// TIA Portal project "Project_Benzinarie" (V15.1)

(* hardware
DEVICE "S71500/ET200MP station_1"  S7-1500 station
   slot 0: "Rail_0"  Rack  6ES7 590-1***0-0AA0
   slot 1: "PLC_1"  CPU 1513-1 PN  6ES7 513-1AL02-0AB0  V2.6
      slot 3: "CPU display_1"  6ES7591-1AA00-0AA0
*)

// ===== PLC "PLC_1"  CPU 1513-1 PN =====

VAR_GLOBAL   // PLC tag table "Default tag table"
   "Clock_Byte" AT %MB0 : Byte;
   "Clock_10Hz" AT %M0.0 : Bool;
   "Clock_5Hz" AT %M0.1 : Bool;
   "Clock_2.5Hz" AT %M0.2 : Bool;
   "Clock_2Hz" AT %M0.3 : Bool;
   "Clock_1.25Hz" AT %M0.4 : Bool;
   "Clock_1Hz" AT %M0.5 : Bool;
   "Clock_0.625Hz" AT %M0.6 : Bool;
   "Clock_0.5Hz" AT %M0.7 : Bool;
END_VAR

DATA_BLOCK "Alarme"   // DB1
{ S7_Optimized_Access := 'TRUE' }
VERSION : 0.1
   VAR
      alarme_gather : Word;
      alarme_vect : Array[0..15] of Bool;
   END_VAR
BEGIN
END_DATA_BLOCK

DATA_BLOCK "Avarii"   // DB2
{ S7_Optimized_Access := 'TRUE' }
VERSION : 0.1
   VAR
      esd : Bool;
      esd_btn : Bool;
      reset_esd : Bool;
      avarie_p1 : Bool;
      avarie_p2 : Bool;
      avarie_p3 : Bool;
      avarie_p4 : Bool;
      reset_avarii : Bool;
   END_VAR
BEGIN
END_DATA_BLOCK

DATA_BLOCK "Bazine"   // DB3
{ S7_Optimized_Access := 'TRUE' }
VERSION : 0.1
   VAR
      benzina_90 : Real;
      benzina_95 : Real;
      motorina : Real;
      motorina_premium : Real;
      "benzina_90_1/2" : Real;
      "benzina_95_1/2" : Real;
      "motorina_1/2" : Real;
      "motorina_premium_1/2" : Real;
      b90_gol : Bool;
      b95_gol : Bool;
      m_gol : Bool;
      m_p_gol : Bool;
      nivel_benzina90 : Real;
      nivel_benzina95 : Real;
      nivel_motorina : Real;
      nivel_motorina_premium : Real;
   END_VAR
BEGIN
END_DATA_BLOCK

DATA_BLOCK "Pompa_benzian90"   // DB4
{ S7_Optimized_Access := 'TRUE' }
VERSION : 0.1
   VAR
      blocare : Bool;
      scoasa : Bool;
      start_clapeta : Bool;
      buton_plata : Bool;
      led_rosu : Bool;
      permisiune_start : Bool;
      index_pret : Real;
      cantitate : Real;
      plata_posibila : Bool;
      terminat : Bool;
      pret : Real;
      nivel_pompa : Real;
      nivel_pompa_iesire : Real;
   END_VAR
BEGIN
END_DATA_BLOCK

DATA_BLOCK "Pompa_benzina95"   // DB5
{ S7_Optimized_Access := 'TRUE' }
VERSION : 0.1
   VAR
      blocare : Bool;
      scoasa : Bool;
      start_clapeta : Bool;
      buton_plata : Bool;
      led_rosu : Bool;
      permisiune_start : Bool;
      index_pret : Real;
      cantitate : Real;
      plata_posibila : Bool;
      terminat : Bool;
      pret : Real;
      nivel_pompa : Real;
      permisiune_pompa : Bool;
   END_VAR
BEGIN
END_DATA_BLOCK

DATA_BLOCK "Pompa_motorina"   // DB6
{ S7_Optimized_Access := 'TRUE' }
VERSION : 0.1
   VAR
      blocare : Bool;
      scoasa : Bool;
      start_clapeta : Bool;
      buton_plata : Bool;
      led_rosu : Bool;
      permisiune_start : Bool;
      index_pret : Real;
      cantitate : Real;
      plata_posibila : Bool;
      terminat : Bool;
      pret : Real;
      nivel_pompa : Real;
      permisiune_pompa : Bool;
   END_VAR
BEGIN
END_DATA_BLOCK

DATA_BLOCK "Pompa_motorina_premium"   // DB7
{ S7_Optimized_Access := 'TRUE' }
VERSION : 0.1
   VAR
      blocare : Bool;
      scoasa : Bool;
      start_clapeta : Bool;
      buton_plata : Bool;
      led_rosu : Bool;
      permisiune_start : Bool;
      index_pret : Real;
      cantitate : Real;
      plata_posibila : Bool;
      terminat : Bool;
      pret : Real;
      nivel_pompa : Real;
      permisiune_pompa : Bool;
   END_VAR
BEGIN
END_DATA_BLOCK

DATA_BLOCK "Benzina90"   // DB8
{ S7_Optimized_Access := 'TRUE' }
VERSION : 0.1
// stored: InstanceOfName Pompa
"Pompa"
BEGIN
END_DATA_BLOCK

DATA_BLOCK "Benzina95"   // DB9
{ S7_Optimized_Access := 'TRUE' }
VERSION : 0.1
// stored: InstanceOfName Pompa
"Pompa"
BEGIN
END_DATA_BLOCK

DATA_BLOCK "Motorina"   // DB10
{ S7_Optimized_Access := 'TRUE' }
VERSION : 0.1
// stored: InstanceOfName Pompa
"Pompa"
BEGIN
END_DATA_BLOCK

DATA_BLOCK "Motorina_premium"   // DB11
{ S7_Optimized_Access := 'TRUE' }
VERSION : 0.1
// stored: InstanceOfName Pompa
"Pompa"
BEGIN
END_DATA_BLOCK

DATA_BLOCK "Butoane_umplere_bazine"   // DB13
{ S7_Optimized_Access := 'TRUE' }
VERSION : 0.1
   VAR
      btn_b90 : Bool;
      btn_b95 : Bool;
      btn_m : Bool;
      btn_m_p : Bool;
   END_VAR
BEGIN
END_DATA_BLOCK

// folder: System blocks/Program resources

DATA_BLOCK "reset_esd"   // DB12
{ S7_Optimized_Access := 'TRUE' }
AUTHOR : Simatic
FAMILY : IEC
NAME : IEC_TMR
VERSION : 1.0
// stored: InstanceOfName IEC_TIMER
"IEC_TIMER"
BEGIN
END_DATA_BLOCK

DATA_BLOCK "reset_avarii"   // DB14
{ S7_Optimized_Access := 'TRUE' }
AUTHOR : Simatic
FAMILY : IEC
NAME : IEC_TMR
VERSION : 1.0
// stored: InstanceOfName IEC_TIMER
"IEC_TIMER"
BEGIN
END_DATA_BLOCK

// folder: (top level)

FUNCTION_BLOCK "Pompa"   // FB1, LAD
{ S7_Optimized_Access := 'TRUE' }
VERSION : 0.1
   VAR_INPUT
      blocare : Bool;
      esd : Bool;
      avarie_interna : Bool;
      bazin_gol : Bool;
   END_VAR
   VAR_OUTPUT
      pret : Real;
      terminat : Bool;
   END_VAR
   VAR_IN_OUT
      scoasa : Bool;
      start_clapeta : Bool;
      bazin : Real;
      buton_plata : Bool;
      led_rosu : Bool;
      permisiune_start : Bool;
      permisiune_pompa : Bool;
      index_pret : Real;
      cantitate : Real;
      plata_posibila : Bool;
      nivel_pompa : Real;
   END_VAR
   VAR
      re1 : Bool;
      re2 : Bool;
      led_intermitent : Bool;
      timer_reset_plata : TON_TIME;
   END_VAR
   VAR_TEMP   // added for the SCL form of the ladder/FBD networks
      _w1 : Bool;
   END_VAR
BEGIN

REGION Network 1: permisiune de start
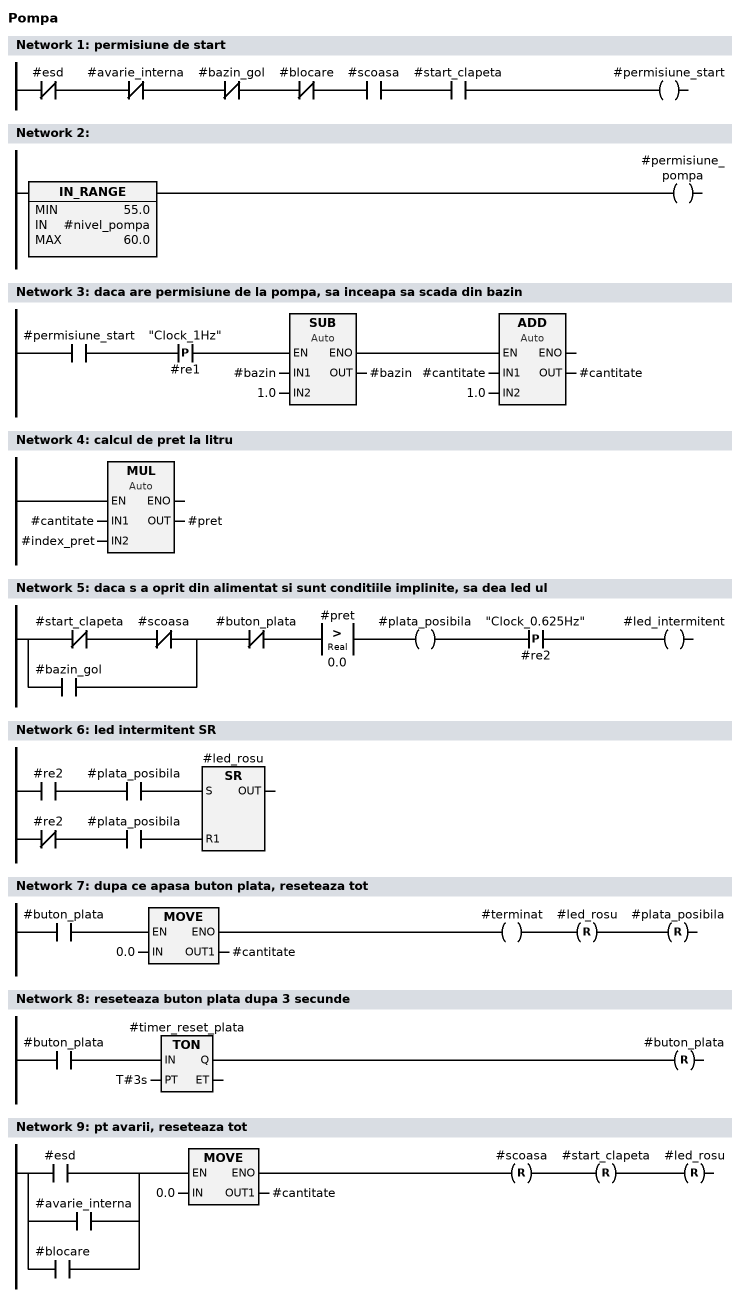
   RUNG wire#powerrail
      I_Contact( #esd )
      I_Contact( #avarie_interna )
      I_Contact( #bazin_gol )
      I_Contact( #blocare )
      Contact( #scoasa )
      Contact( #start_clapeta )
      Coil( #permisiune_start )
   END_RUNG
   // the same network as SCL:
   #permisiune_start := NOT #esd AND NOT #avarie_interna AND NOT #bazin_gol AND NOT #blocare AND #scoasa AND #start_clapeta;
END_REGION

REGION Network 2
   RUNG wire#powerrail
      { S7_Templates := "SrcType := Real" } InRange(min := 55.0, in := #nivel_pompa, max := 60.0)
      Coil( #permisiune_pompa )
   END_RUNG
   // the same network as SCL:
   #permisiune_pompa := (55.0 <= #nivel_pompa) AND (#nivel_pompa <= 60.0);
END_REGION

REGION Network 3: daca are permisiune de la pompa, sa inceapa sa scada din bazin
   RUNG wire#powerrail
      Contact( #permisiune_start )
      P_Contact(operand := "Clock_1Hz", bit := #re1)
      Sub(in1 := #bazin, in2 := 1.0, out => #bazin)
      Add(in1 := #cantitate, in2 := 1.0, out => #cantitate)
   END_RUNG
   // the same network as SCL:
   #_w1 := #permisiune_start AND "Clock_1Hz" AND NOT #re1;   // rising edge of "Clock_1Hz"
   #re1 := "Clock_1Hz";
   IF #_w1 THEN
       #bazin := #bazin - 1.0;
       #cantitate := #cantitate + 1.0;
   END_IF;
END_REGION

REGION Network 4: calcul de pret la litru
   RUNG wire#powerrail
      Mul(in1 := #cantitate, in2 := #index_pret, out => #pret)
   END_RUNG
   // the same network as SCL:
   #pret := #cantitate * #index_pret;
END_REGION

REGION Network 5: daca s a oprit din alimentat si sunt conditiile implinite, sa dea led ul
   RUNG wire#powerrail
      I_Contact( #start_clapeta )
      I_Contact( #scoasa )
      wire#w1
      I_Contact( #buton_plata )
      { S7_Templates := "SrcType := Real" } GT_Contact(in1 := #pret, in2 := 0.0)
      Coil( #plata_posibila )
      P_Contact(operand := "Clock_0.625Hz", bit := #re2)
      Coil( #led_intermitent )
   END_RUNG
   RUNG wire#powerrail
      Contact( #bazin_gol )
   END_RUNG wire#w1
   // the same network as SCL:
   #plata_posibila := ((NOT #start_clapeta AND NOT #scoasa) OR #bazin_gol) AND NOT #buton_plata AND (#pret > 0.0);
   #_w1 := #plata_posibila AND "Clock_0.625Hz" AND NOT #re2;   // rising edge of "Clock_0.625Hz"
   #re2 := "Clock_0.625Hz";
   #led_intermitent := #_w1;
END_REGION

REGION Network 6: led intermitent SR
   RUNG wire#powerrail
      Contact( #re2 )
      Contact( #plata_posibila )
      S_SR(operand := #led_rosu, r1 := wire#w1)
   END_RUNG
   RUNG wire#powerrail
      I_Contact( #re2 )
      Contact( #plata_posibila )
   END_RUNG wire#w1
   // the same network as SCL:
   IF #re2 AND #plata_posibila THEN
       #led_rosu := TRUE;   // SR flip-flop
   END_IF;
   IF NOT #re2 AND #plata_posibila THEN #led_rosu := FALSE; END_IF;
END_REGION

REGION Network 7: dupa ce apasa buton plata, reseteaza tot
   RUNG wire#powerrail
      Contact( #buton_plata )
      Move(in := 0.0, out1 => #cantitate)
      Coil( #terminat )
      R_Coil( #led_rosu )
      R_Coil( #plata_posibila )
   END_RUNG
   // the same network as SCL:
   IF #buton_plata THEN #cantitate := 0.0; END_IF;
   #terminat := #buton_plata;
   IF #buton_plata THEN
       #led_rosu := FALSE;
       #plata_posibila := FALSE;
   END_IF;
END_REGION

REGION Network 8: reseteaza buton plata dupa 3 secunde
   #timer_reset_plata(IN := #buton_plata, PT := T#3s);   // TON
   IF #timer_reset_plata.Q THEN #buton_plata := FALSE; END_IF;
END_REGION

REGION Network 9: pt avarii, reseteaza tot
   RUNG wire#powerrail
      Contact( #esd )
      wire#w1
      Move(in := 0.0, out1 => #cantitate)
      R_Coil( #scoasa )
      R_Coil( #start_clapeta )
      R_Coil( #led_rosu )
   END_RUNG
   RUNG wire#powerrail
      Contact( #avarie_interna )
   END_RUNG wire#w1
   RUNG wire#powerrail
      Contact( #blocare )
   END_RUNG wire#w1
   // the same network as SCL:
   IF #esd OR #avarie_interna OR #blocare THEN
       #cantitate := 0.0;
       #scoasa := FALSE;
       #start_clapeta := FALSE;
       #led_rosu := FALSE;
   END_IF;
END_REGION
END_FUNCTION_BLOCK

ORGANIZATION_BLOCK "Main"   // OB1, LAD, ProgramCycle
TITLE = "Main Program Sweep (Cycle)"
{ S7_Optimized_Access := 'TRUE' }
VERSION : 0.1
   VAR_INPUT
      Initial_Call : Bool;   // Initial call of this OB
      Remanence : Bool;   // =True, if remanent data are available
   END_VAR
   VAR_TEMP   // added for the SCL form of the ladder/FBD networks
      _w1 : Bool;
      _w2 : Bool;
      _w3 : Bool;
      _w4 : Bool;
   END_VAR
BEGIN

REGION Network 1: benzina90
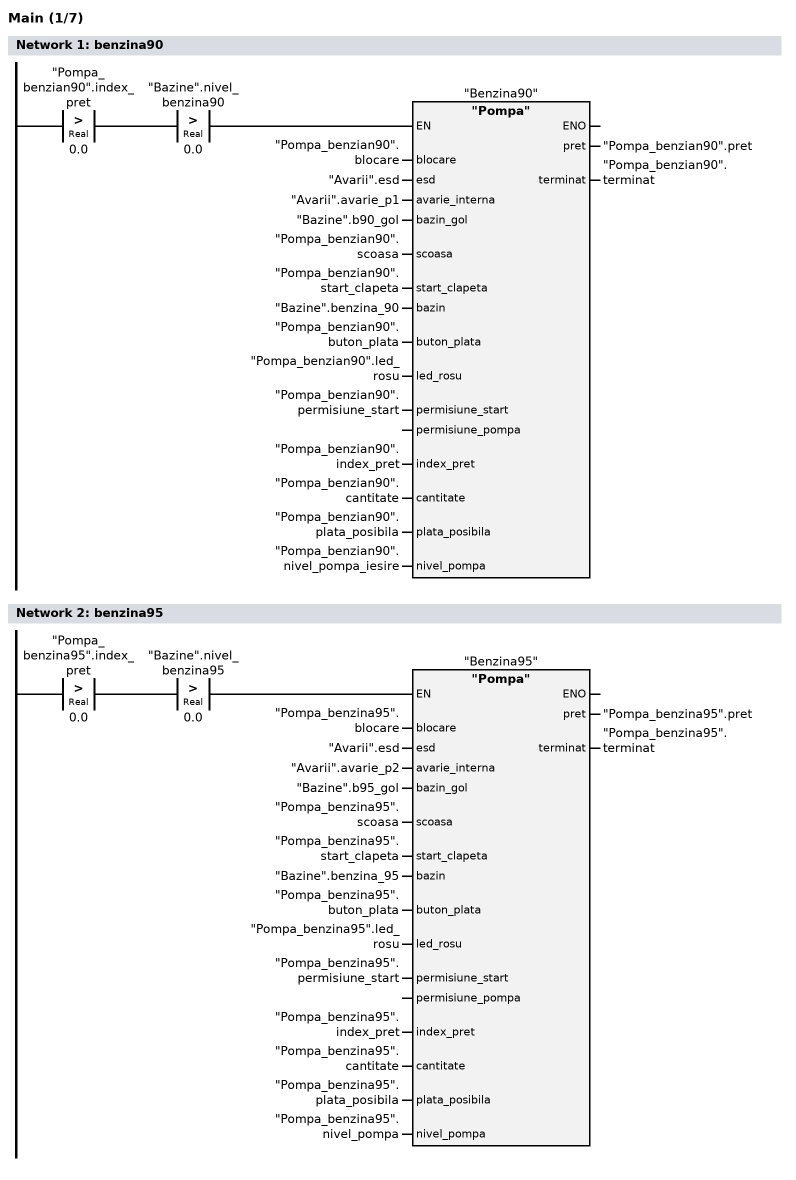
   RUNG wire#powerrail
      { S7_Templates := "SrcType := Real" } GT_Contact(in1 := "Pompa_benzian90".index_pret, in2 := 0.0)
      { S7_Templates := "SrcType := Real" } GT_Contact(in1 := "Bazine".nivel_benzina90, in2 := 0.0)
      "Benzina90"(blocare := "Pompa_benzian90".blocare, esd := "Avarii".esd, avarie_interna := "Avarii".avarie_p1, bazin_gol := "Bazine".b90_gol, scoasa := "Pompa_benzian90".scoasa, start_clapeta := "Pompa_benzian90".start_clapeta, bazin := "Bazine".benzina_90, buton_plata := "Pompa_benzian90".buton_plata, led_rosu := "Pompa_benzian90".led_rosu, permisiune_start := "Pompa_benzian90".permisiune_start, permisiune_pompa :=, index_pret := "Pompa_benzian90".index_pret, cantitate := "Pompa_benzian90".cantitate, plata_posibila := "Pompa_benzian90".plata_posibila, nivel_pompa := "Pompa_benzian90".nivel_pompa_iesire, pret => "Pompa_benzian90".pret, terminat => "Pompa_benzian90".terminat)
   END_RUNG
   // the same network as SCL:
   IF ("Pompa_benzian90".index_pret > 0.0) AND ("Bazine".nivel_benzina90 > 0.0) THEN
       "Benzina90"(blocare := "Pompa_benzian90".blocare,   // "Pompa"
                   esd := "Avarii".esd,
                   avarie_interna := "Avarii".avarie_p1,
                   bazin_gol := "Bazine".b90_gol,
                   scoasa := "Pompa_benzian90".scoasa,
                   start_clapeta := "Pompa_benzian90".start_clapeta,
                   bazin := "Bazine".benzina_90,
                   buton_plata := "Pompa_benzian90".buton_plata,
                   led_rosu := "Pompa_benzian90".led_rosu,
                   permisiune_start := "Pompa_benzian90".permisiune_start,
                   index_pret := "Pompa_benzian90".index_pret,
                   cantitate := "Pompa_benzian90".cantitate,
                   plata_posibila := "Pompa_benzian90".plata_posibila,
                   nivel_pompa := "Pompa_benzian90".nivel_pompa_iesire,
                   pret => "Pompa_benzian90".pret,
                   terminat => "Pompa_benzian90".terminat);
   END_IF;
END_REGION

REGION Network 2: benzina95
   RUNG wire#powerrail
      { S7_Templates := "SrcType := Real" } GT_Contact(in1 := "Pompa_benzina95".index_pret, in2 := 0.0)
      { S7_Templates := "SrcType := Real" } GT_Contact(in1 := "Bazine".nivel_benzina95, in2 := 0.0)
      "Benzina95"(blocare := "Pompa_benzina95".blocare, esd := "Avarii".esd, avarie_interna := "Avarii".avarie_p2, bazin_gol := "Bazine".b95_gol, scoasa := "Pompa_benzina95".scoasa, start_clapeta := "Pompa_benzina95".start_clapeta, bazin := "Bazine".benzina_95, buton_plata := "Pompa_benzina95".buton_plata, led_rosu := "Pompa_benzina95".led_rosu, permisiune_start := "Pompa_benzina95".permisiune_start, permisiune_pompa :=, index_pret := "Pompa_benzina95".index_pret, cantitate := "Pompa_benzina95".cantitate, plata_posibila := "Pompa_benzina95".plata_posibila, nivel_pompa := "Pompa_benzina95".nivel_pompa, pret => "Pompa_benzina95".pret, terminat => "Pompa_benzina95".terminat)
   END_RUNG
   // the same network as SCL:
   IF ("Pompa_benzina95".index_pret > 0.0) AND ("Bazine".nivel_benzina95 > 0.0) THEN
       "Benzina95"(blocare := "Pompa_benzina95".blocare,   // "Pompa"
                   esd := "Avarii".esd,
                   avarie_interna := "Avarii".avarie_p2,
                   bazin_gol := "Bazine".b95_gol,
                   scoasa := "Pompa_benzina95".scoasa,
                   start_clapeta := "Pompa_benzina95".start_clapeta,
                   bazin := "Bazine".benzina_95,
                   buton_plata := "Pompa_benzina95".buton_plata,
                   led_rosu := "Pompa_benzina95".led_rosu,
                   permisiune_start := "Pompa_benzina95".permisiune_start,
                   index_pret := "Pompa_benzina95".index_pret,
                   cantitate := "Pompa_benzina95".cantitate,
                   plata_posibila := "Pompa_benzina95".plata_posibila,
                   nivel_pompa := "Pompa_benzina95".nivel_pompa,
                   pret => "Pompa_benzina95".pret,
                   terminat => "Pompa_benzina95".terminat);
   END_IF;
END_REGION

REGION Network 3: motorina
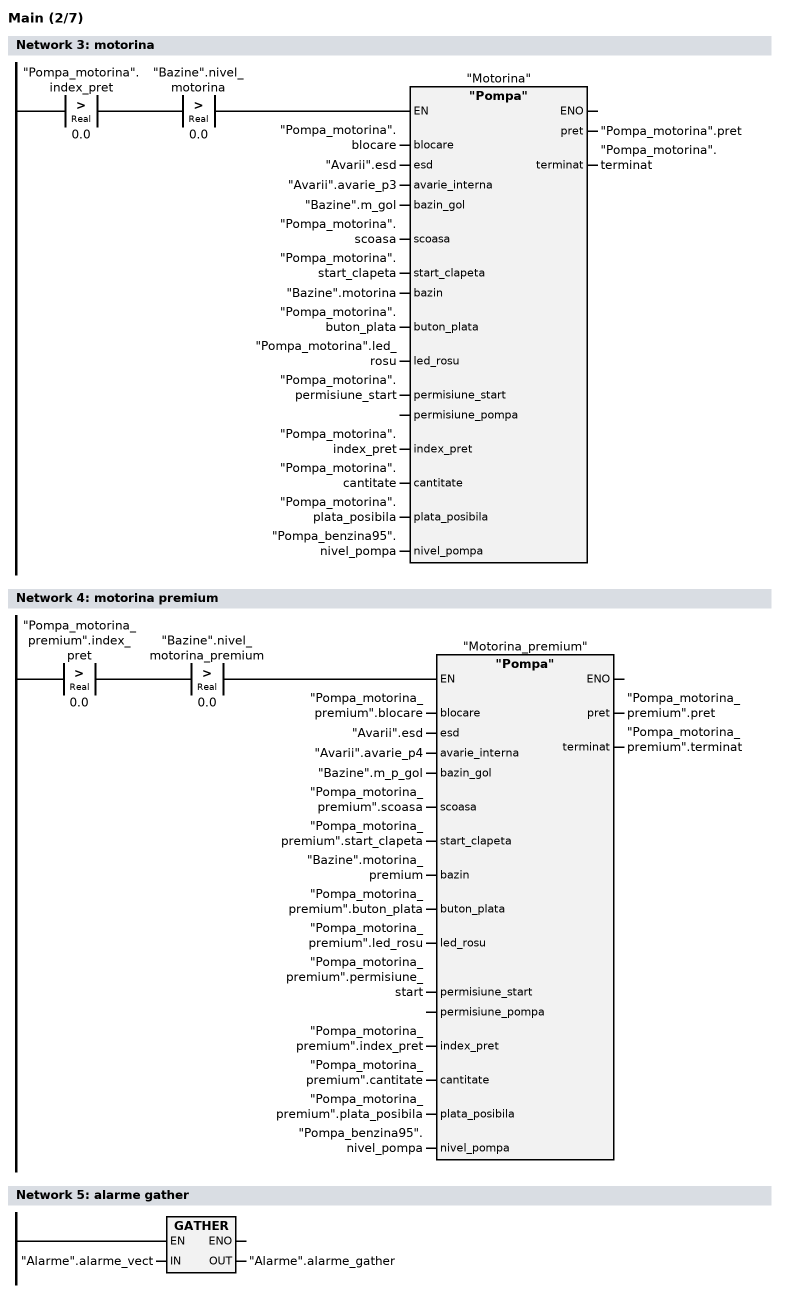
   RUNG wire#powerrail
      { S7_Templates := "SrcType := Real" } GT_Contact(in1 := "Pompa_motorina".index_pret, in2 := 0.0)
      { S7_Templates := "SrcType := Real" } GT_Contact(in1 := "Bazine".nivel_motorina, in2 := 0.0)
      "Motorina"(blocare := "Pompa_motorina".blocare, esd := "Avarii".esd, avarie_interna := "Avarii".avarie_p3, bazin_gol := "Bazine".m_gol, scoasa := "Pompa_motorina".scoasa, start_clapeta := "Pompa_motorina".start_clapeta, bazin := "Bazine".motorina, buton_plata := "Pompa_motorina".buton_plata, led_rosu := "Pompa_motorina".led_rosu, permisiune_start := "Pompa_motorina".permisiune_start, permisiune_pompa :=, index_pret := "Pompa_motorina".index_pret, cantitate := "Pompa_motorina".cantitate, plata_posibila := "Pompa_motorina".plata_posibila, nivel_pompa := "Pompa_benzina95".nivel_pompa, pret => "Pompa_motorina".pret, terminat => "Pompa_motorina".terminat)
   END_RUNG
   // the same network as SCL:
   IF ("Pompa_motorina".index_pret > 0.0) AND ("Bazine".nivel_motorina > 0.0) THEN
       "Motorina"(blocare := "Pompa_motorina".blocare,   // "Pompa"
                  esd := "Avarii".esd,
                  avarie_interna := "Avarii".avarie_p3,
                  bazin_gol := "Bazine".m_gol,
                  scoasa := "Pompa_motorina".scoasa,
                  start_clapeta := "Pompa_motorina".start_clapeta,
                  bazin := "Bazine".motorina,
                  buton_plata := "Pompa_motorina".buton_plata,
                  led_rosu := "Pompa_motorina".led_rosu,
                  permisiune_start := "Pompa_motorina".permisiune_start,
                  index_pret := "Pompa_motorina".index_pret,
                  cantitate := "Pompa_motorina".cantitate,
                  plata_posibila := "Pompa_motorina".plata_posibila,
                  nivel_pompa := "Pompa_benzina95".nivel_pompa,
                  pret => "Pompa_motorina".pret,
                  terminat => "Pompa_motorina".terminat);
   END_IF;
END_REGION

REGION Network 4: motorina premium
   RUNG wire#powerrail
      { S7_Templates := "SrcType := Real" } GT_Contact(in1 := "Pompa_motorina_premium".index_pret, in2 := 0.0)
      { S7_Templates := "SrcType := Real" } GT_Contact(in1 := "Bazine".nivel_motorina_premium, in2 := 0.0)
      "Motorina_premium"(blocare := "Pompa_motorina_premium".blocare, esd := "Avarii".esd, avarie_interna := "Avarii".avarie_p4, bazin_gol := "Bazine".m_p_gol, scoasa := "Pompa_motorina_premium".scoasa, start_clapeta := "Pompa_motorina_premium".start_clapeta, bazin := "Bazine".motorina_premium, buton_plata := "Pompa_motorina_premium".buton_plata, led_rosu := "Pompa_motorina_premium".led_rosu, permisiune_start := "Pompa_motorina_premium".permisiune_start, permisiune_pompa :=, index_pret := "Pompa_motorina_premium".index_pret, cantitate := "Pompa_motorina_premium".cantitate, plata_posibila := "Pompa_motorina_premium".plata_posibila, nivel_pompa := "Pompa_benzina95".nivel_pompa, pret => "Pompa_motorina_premium".pret, terminat => "Pompa_motorina_premium".terminat)
   END_RUNG
   // the same network as SCL:
   IF ("Pompa_motorina_premium".index_pret > 0.0) AND ("Bazine".nivel_motorina_premium > 0.0) THEN
       "Motorina_premium"(blocare := "Pompa_motorina_premium".blocare,   // "Pompa"
                          esd := "Avarii".esd,
                          avarie_interna := "Avarii".avarie_p4,
                          bazin_gol := "Bazine".m_p_gol,
                          scoasa := "Pompa_motorina_premium".scoasa,
                          start_clapeta := "Pompa_motorina_premium".start_clapeta,
                          bazin := "Bazine".motorina_premium,
                          buton_plata := "Pompa_motorina_premium".buton_plata,
                          led_rosu := "Pompa_motorina_premium".led_rosu,
                          permisiune_start := "Pompa_motorina_premium".permisiune_start,
                          index_pret := "Pompa_motorina_premium".index_pret,
                          cantitate := "Pompa_motorina_premium".cantitate,
                          plata_posibila := "Pompa_motorina_premium".plata_posibila,
                          nivel_pompa := "Pompa_benzina95".nivel_pompa,
                          pret => "Pompa_motorina_premium".pret,
                          terminat => "Pompa_motorina_premium".terminat);
   END_IF;
END_REGION

REGION Network 5: alarme gather
   GATHER(IN := "Alarme".alarme_vect, OUT => "Alarme".alarme_gather);
END_REGION

REGION Network 6: umplere bazin la maxim cand e apasat butonul
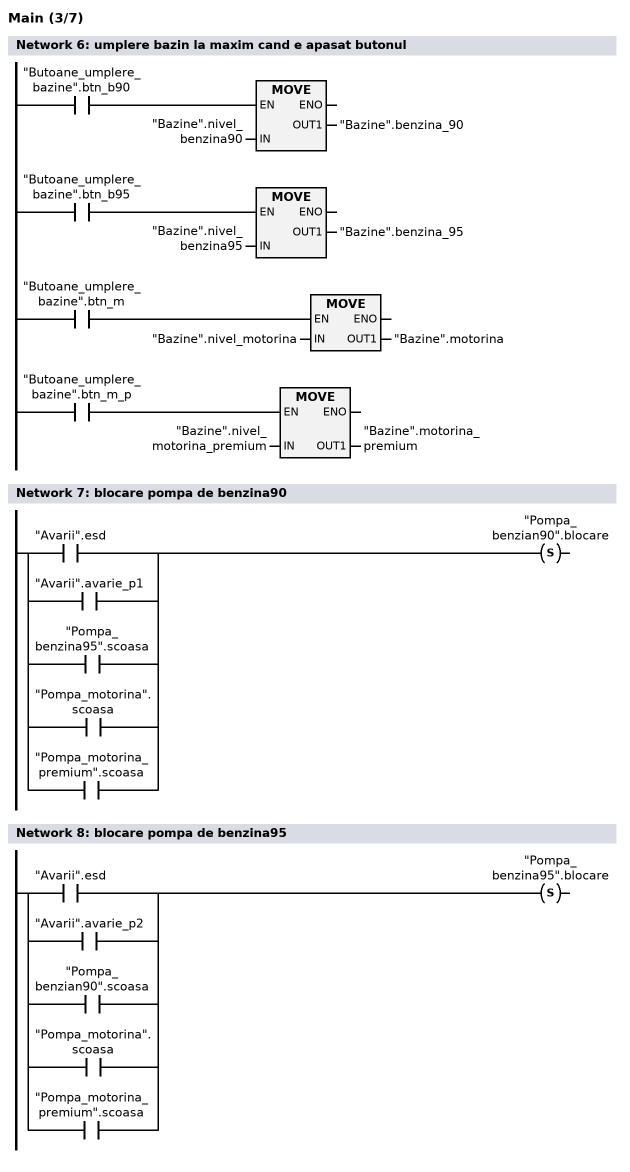
   RUNG wire#powerrail
      Contact( "Butoane_umplere_bazine".btn_b90 )
      Move(in := "Bazine".nivel_benzina90, out1 => "Bazine".benzina_90)
   END_RUNG
   RUNG wire#powerrail
      Contact( "Butoane_umplere_bazine".btn_b95 )
      Move(in := "Bazine".nivel_benzina95, out1 => "Bazine".benzina_95)
   END_RUNG
   RUNG wire#powerrail
      Contact( "Butoane_umplere_bazine".btn_m )
      Move(in := "Bazine".nivel_motorina, out1 => "Bazine".motorina)
   END_RUNG
   RUNG wire#powerrail
      Contact( "Butoane_umplere_bazine".btn_m_p )
      Move(in := "Bazine".nivel_motorina_premium, out1 => "Bazine".motorina_premium)
   END_RUNG
   // the same network as SCL:
   IF "Butoane_umplere_bazine".btn_b90 THEN "Bazine".benzina_90 := "Bazine".nivel_benzina90; END_IF;
   IF "Butoane_umplere_bazine".btn_b95 THEN "Bazine".benzina_95 := "Bazine".nivel_benzina95; END_IF;
   IF "Butoane_umplere_bazine".btn_m THEN "Bazine".motorina := "Bazine".nivel_motorina; END_IF;
   IF "Butoane_umplere_bazine".btn_m_p THEN
       "Bazine".motorina_premium := "Bazine".nivel_motorina_premium;
   END_IF;
END_REGION

REGION Network 7: blocare pompa de benzina90
   RUNG wire#powerrail
      Contact( "Avarii".esd )
      wire#w1
      S_Coil( "Pompa_benzian90".blocare )
   END_RUNG
   RUNG wire#powerrail
      Contact( "Avarii".avarie_p1 )
   END_RUNG wire#w1
   RUNG wire#powerrail
      Contact( "Pompa_benzina95".scoasa )
   END_RUNG wire#w1
   RUNG wire#powerrail
      Contact( "Pompa_motorina".scoasa )
   END_RUNG wire#w1
   RUNG wire#powerrail
      Contact( "Pompa_motorina_premium".scoasa )
   END_RUNG wire#w1
   // the same network as SCL:
   IF "Avarii".esd OR "Avarii".avarie_p1 OR "Pompa_benzina95".scoasa OR "Pompa_motorina".scoasa OR "Pompa_motorina_premium".scoasa THEN
       "Pompa_benzian90".blocare := TRUE;
   END_IF;
END_REGION

REGION Network 8: blocare pompa de benzina95
   RUNG wire#powerrail
      Contact( "Avarii".esd )
      wire#w1
      S_Coil( "Pompa_benzina95".blocare )
   END_RUNG
   RUNG wire#powerrail
      Contact( "Avarii".avarie_p2 )
   END_RUNG wire#w1
   RUNG wire#powerrail
      Contact( "Pompa_benzian90".scoasa )
   END_RUNG wire#w1
   RUNG wire#powerrail
      Contact( "Pompa_motorina".scoasa )
   END_RUNG wire#w1
   RUNG wire#powerrail
      Contact( "Pompa_motorina_premium".scoasa )
   END_RUNG wire#w1
   // the same network as SCL:
   IF "Avarii".esd OR "Avarii".avarie_p2 OR "Pompa_benzian90".scoasa OR "Pompa_motorina".scoasa OR "Pompa_motorina_premium".scoasa THEN
       "Pompa_benzina95".blocare := TRUE;
   END_IF;
END_REGION

REGION Network 9: blocare pompa de motorina
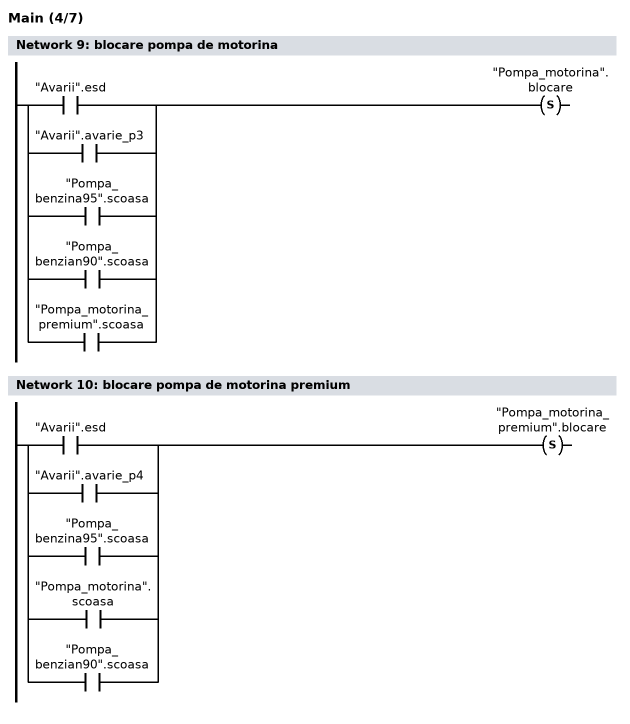
   RUNG wire#powerrail
      Contact( "Avarii".esd )
      wire#w1
      S_Coil( "Pompa_motorina".blocare )
   END_RUNG
   RUNG wire#powerrail
      Contact( "Avarii".avarie_p3 )
   END_RUNG wire#w1
   RUNG wire#powerrail
      Contact( "Pompa_benzina95".scoasa )
   END_RUNG wire#w1
   RUNG wire#powerrail
      Contact( "Pompa_benzian90".scoasa )
   END_RUNG wire#w1
   RUNG wire#powerrail
      Contact( "Pompa_motorina_premium".scoasa )
   END_RUNG wire#w1
   // the same network as SCL:
   IF "Avarii".esd OR "Avarii".avarie_p3 OR "Pompa_benzina95".scoasa OR "Pompa_benzian90".scoasa OR "Pompa_motorina_premium".scoasa THEN
       "Pompa_motorina".blocare := TRUE;
   END_IF;
END_REGION

REGION Network 10: blocare pompa de motorina premium
   RUNG wire#powerrail
      Contact( "Avarii".esd )
      wire#w1
      S_Coil( "Pompa_motorina_premium".blocare )
   END_RUNG
   RUNG wire#powerrail
      Contact( "Avarii".avarie_p4 )
   END_RUNG wire#w1
   RUNG wire#powerrail
      Contact( "Pompa_benzina95".scoasa )
   END_RUNG wire#w1
   RUNG wire#powerrail
      Contact( "Pompa_motorina".scoasa )
   END_RUNG wire#w1
   RUNG wire#powerrail
      Contact( "Pompa_benzian90".scoasa )
   END_RUNG wire#w1
   // the same network as SCL:
   IF "Avarii".esd OR "Avarii".avarie_p4 OR "Pompa_benzina95".scoasa OR "Pompa_motorina".scoasa OR "Pompa_benzian90".scoasa THEN
       "Pompa_motorina_premium".blocare := TRUE;
   END_IF;
END_REGION

REGION Network 11: reseteaza blocarea la pompe daca se termina
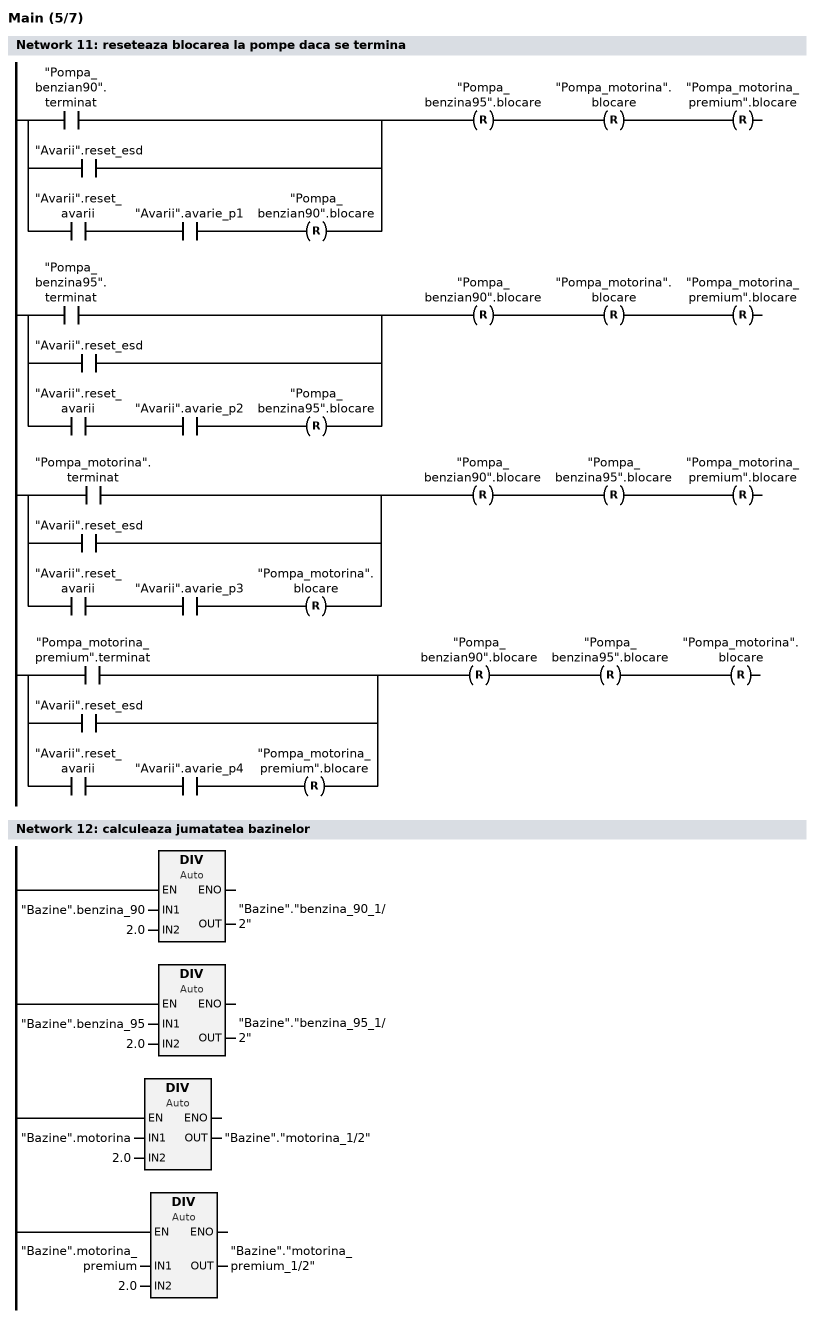
   RUNG wire#powerrail
      Contact( "Pompa_benzian90".terminat )
      wire#w1
      R_Coil( "Pompa_benzina95".blocare )
      R_Coil( "Pompa_motorina".blocare )
      R_Coil( "Pompa_motorina_premium".blocare )
   END_RUNG
   RUNG wire#powerrail
      Contact( "Avarii".reset_esd )
   END_RUNG wire#w1
   RUNG wire#powerrail
      Contact( "Avarii".reset_avarii )
      Contact( "Avarii".avarie_p1 )
      R_Coil( "Pompa_benzian90".blocare )
   END_RUNG wire#w1
   RUNG wire#powerrail
      Contact( "Pompa_benzina95".terminat )
      wire#w2
      R_Coil( "Pompa_benzian90".blocare )
      R_Coil( "Pompa_motorina".blocare )
      R_Coil( "Pompa_motorina_premium".blocare )
   END_RUNG
   RUNG wire#powerrail
      Contact( "Avarii".reset_esd )
   END_RUNG wire#w2
   RUNG wire#powerrail
      Contact( "Avarii".reset_avarii )
      Contact( "Avarii".avarie_p2 )
      R_Coil( "Pompa_benzina95".blocare )
   END_RUNG wire#w2
   RUNG wire#powerrail
      Contact( "Pompa_motorina".terminat )
      wire#w3
      R_Coil( "Pompa_benzian90".blocare )
      R_Coil( "Pompa_benzina95".blocare )
      R_Coil( "Pompa_motorina_premium".blocare )
   END_RUNG
   RUNG wire#powerrail
      Contact( "Avarii".reset_esd )
   END_RUNG wire#w3
   RUNG wire#powerrail
      Contact( "Avarii".reset_avarii )
      Contact( "Avarii".avarie_p3 )
      R_Coil( "Pompa_motorina".blocare )
   END_RUNG wire#w3
   RUNG wire#powerrail
      Contact( "Pompa_motorina_premium".terminat )
      wire#w4
      R_Coil( "Pompa_benzian90".blocare )
      R_Coil( "Pompa_benzina95".blocare )
      R_Coil( "Pompa_motorina".blocare )
   END_RUNG
   RUNG wire#powerrail
      Contact( "Avarii".reset_esd )
   END_RUNG wire#w4
   RUNG wire#powerrail
      Contact( "Avarii".reset_avarii )
      Contact( "Avarii".avarie_p4 )
      R_Coil( "Pompa_motorina_premium".blocare )
   END_RUNG wire#w4
   // the same network as SCL:
   #_w1 := "Avarii".reset_avarii AND "Avarii".avarie_p1;
   IF #_w1 THEN "Pompa_benzian90".blocare := FALSE; END_IF;
   IF "Pompa_benzian90".terminat OR "Avarii".reset_esd OR #_w1 THEN
       "Pompa_benzina95".blocare := FALSE;
       "Pompa_motorina".blocare := FALSE;
       "Pompa_motorina_premium".blocare := FALSE;
   END_IF;
   #_w2 := "Avarii".reset_avarii AND "Avarii".avarie_p2;
   IF #_w2 THEN "Pompa_benzina95".blocare := FALSE; END_IF;
   IF "Pompa_benzina95".terminat OR "Avarii".reset_esd OR #_w2 THEN
       "Pompa_benzian90".blocare := FALSE;
       "Pompa_motorina".blocare := FALSE;
       "Pompa_motorina_premium".blocare := FALSE;
   END_IF;
   #_w3 := "Avarii".reset_avarii AND "Avarii".avarie_p3;
   IF #_w3 THEN "Pompa_motorina".blocare := FALSE; END_IF;
   IF "Pompa_motorina".terminat OR "Avarii".reset_esd OR #_w3 THEN
       "Pompa_benzian90".blocare := FALSE;
       "Pompa_benzina95".blocare := FALSE;
       "Pompa_motorina_premium".blocare := FALSE;
   END_IF;
   #_w4 := "Avarii".reset_avarii AND "Avarii".avarie_p4;
   IF #_w4 THEN "Pompa_motorina_premium".blocare := FALSE; END_IF;
   IF "Pompa_motorina_premium".terminat OR "Avarii".reset_esd OR #_w4 THEN
       "Pompa_benzian90".blocare := FALSE;
       "Pompa_benzina95".blocare := FALSE;
       "Pompa_motorina".blocare := FALSE;
   END_IF;
END_REGION

REGION Network 12: calculeaza jumatatea bazinelor
   RUNG wire#powerrail
      Div(in1 := "Bazine".benzina_90, in2 := 2.0, out => "Bazine"."benzina_90_1/2")
   END_RUNG
   RUNG wire#powerrail
      Div(in1 := "Bazine".benzina_95, in2 := 2.0, out => "Bazine"."benzina_95_1/2")
   END_RUNG
   RUNG wire#powerrail
      Div(in1 := "Bazine".motorina, in2 := 2.0, out => "Bazine"."motorina_1/2")
   END_RUNG
   RUNG wire#powerrail
      Div(in1 := "Bazine".motorina_premium, in2 := 2.0, out => "Bazine"."motorina_premium_1/2")
   END_RUNG
   // the same network as SCL:
   "Bazine"."benzina_90_1/2" := "Bazine".benzina_90 / 2.0;
   "Bazine"."benzina_95_1/2" := "Bazine".benzina_95 / 2.0;
   "Bazine"."motorina_1/2" := "Bazine".motorina / 2.0;
   "Bazine"."motorina_premium_1/2" := "Bazine".motorina_premium / 2.0;
END_REGION

REGION Network 13: bazin la jumate
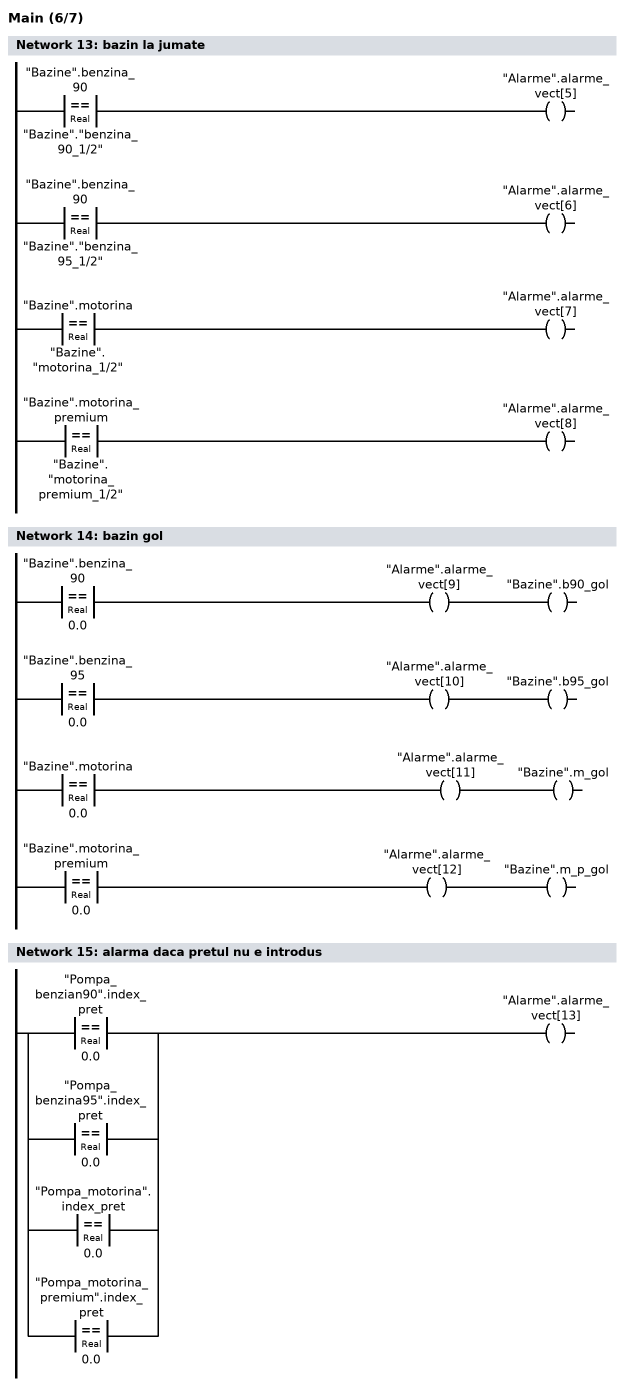
   RUNG wire#powerrail
      { S7_Templates := "SrcType := Real" } EQ_Contact(in1 := "Bazine".benzina_90, in2 := "Bazine"."benzina_90_1/2")
      Coil( "Alarme".alarme_vect[5] )
   END_RUNG
   RUNG wire#powerrail
      { S7_Templates := "SrcType := Real" } EQ_Contact(in1 := "Bazine".benzina_90, in2 := "Bazine"."benzina_95_1/2")
      Coil( "Alarme".alarme_vect[6] )
   END_RUNG
   RUNG wire#powerrail
      { S7_Templates := "SrcType := Real" } EQ_Contact(in1 := "Bazine".motorina, in2 := "Bazine"."motorina_1/2")
      Coil( "Alarme".alarme_vect[7] )
   END_RUNG
   RUNG wire#powerrail
      { S7_Templates := "SrcType := Real" } EQ_Contact(in1 := "Bazine".motorina_premium, in2 := "Bazine"."motorina_premium_1/2")
      Coil( "Alarme".alarme_vect[8] )
   END_RUNG
   // the same network as SCL:
   "Alarme".alarme_vect[5] := "Bazine".benzina_90 = "Bazine"."benzina_90_1/2";
   "Alarme".alarme_vect[6] := "Bazine".benzina_90 = "Bazine"."benzina_95_1/2";
   "Alarme".alarme_vect[7] := "Bazine".motorina = "Bazine"."motorina_1/2";
   "Alarme".alarme_vect[8] := "Bazine".motorina_premium = "Bazine"."motorina_premium_1/2";
END_REGION

REGION Network 14: bazin gol
   RUNG wire#powerrail
      { S7_Templates := "SrcType := Real" } EQ_Contact(in1 := "Bazine".benzina_90, in2 := 0.0)
      Coil( "Alarme".alarme_vect[9] )
      Coil( "Bazine".b90_gol )
   END_RUNG
   RUNG wire#powerrail
      { S7_Templates := "SrcType := Real" } EQ_Contact(in1 := "Bazine".benzina_95, in2 := 0.0)
      Coil( "Alarme".alarme_vect[10] )
      Coil( "Bazine".b95_gol )
   END_RUNG
   RUNG wire#powerrail
      { S7_Templates := "SrcType := Real" } EQ_Contact(in1 := "Bazine".motorina, in2 := 0.0)
      Coil( "Alarme".alarme_vect[11] )
      Coil( "Bazine".m_gol )
   END_RUNG
   RUNG wire#powerrail
      { S7_Templates := "SrcType := Real" } EQ_Contact(in1 := "Bazine".motorina_premium, in2 := 0.0)
      Coil( "Alarme".alarme_vect[12] )
      Coil( "Bazine".m_p_gol )
   END_RUNG
   // the same network as SCL:
   "Alarme".alarme_vect[9] := "Bazine".benzina_90 = 0.0;
   "Bazine".b90_gol := "Bazine".benzina_90 = 0.0;
   "Alarme".alarme_vect[10] := "Bazine".benzina_95 = 0.0;
   "Bazine".b95_gol := "Bazine".benzina_95 = 0.0;
   "Alarme".alarme_vect[11] := "Bazine".motorina = 0.0;
   "Bazine".m_gol := "Bazine".motorina = 0.0;
   "Alarme".alarme_vect[12] := "Bazine".motorina_premium = 0.0;
   "Bazine".m_p_gol := "Bazine".motorina_premium = 0.0;
END_REGION

REGION Network 15: alarma daca pretul nu e introdus
   RUNG wire#powerrail
      { S7_Templates := "SrcType := Real" } EQ_Contact(in1 := "Pompa_benzian90".index_pret, in2 := 0.0)
      wire#w1
      Coil( "Alarme".alarme_vect[13] )
   END_RUNG
   RUNG wire#powerrail
      { S7_Templates := "SrcType := Real" } EQ_Contact(in1 := "Pompa_benzina95".index_pret, in2 := 0.0)
   END_RUNG wire#w1
   RUNG wire#powerrail
      { S7_Templates := "SrcType := Real" } EQ_Contact(in1 := "Pompa_motorina".index_pret, in2 := 0.0)
   END_RUNG wire#w1
   RUNG wire#powerrail
      { S7_Templates := "SrcType := Real" } EQ_Contact(in1 := "Pompa_motorina_premium".index_pret, in2 := 0.0)
   END_RUNG wire#w1
   // the same network as SCL:
   "Alarme".alarme_vect[13] := ("Pompa_benzian90".index_pret = 0.0) OR ("Pompa_benzina95".index_pret = 0.0) OR ("Pompa_motorina".index_pret = 0.0) OR ("Pompa_motorina_premium".index_pret = 0.0);
END_REGION

REGION Network 16: alarma daca bazinelenu au capacitatea introdusa
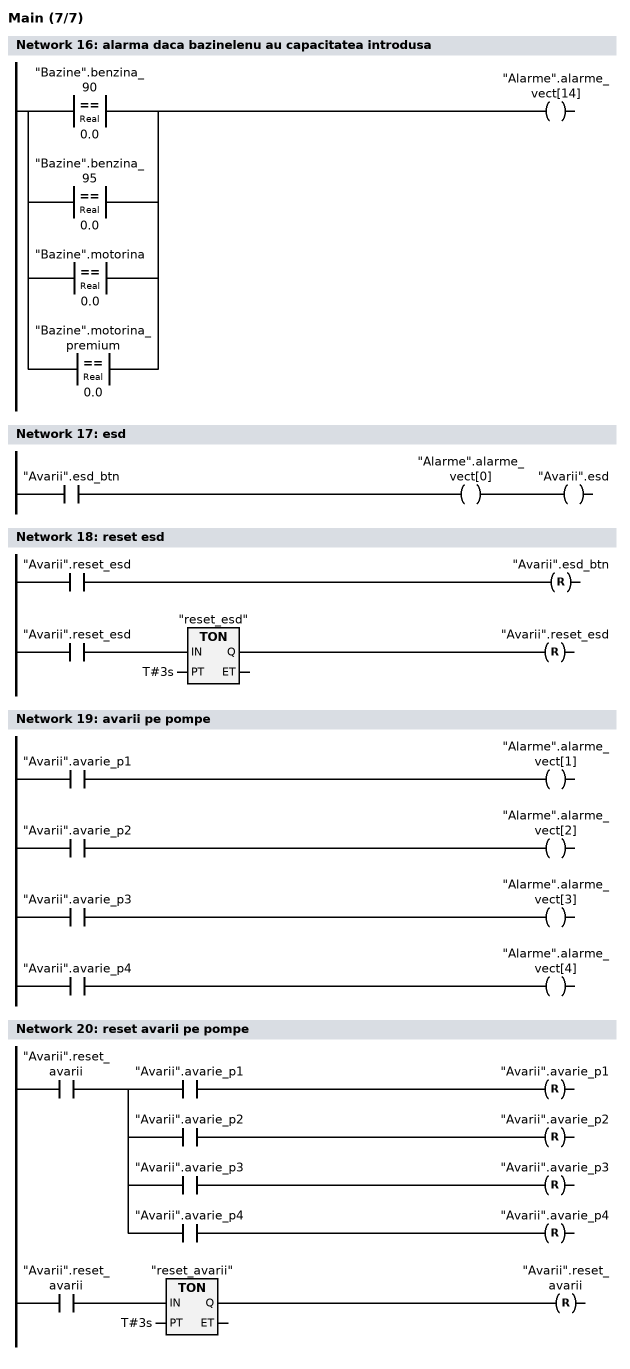
   RUNG wire#powerrail
      { S7_Templates := "SrcType := Real" } EQ_Contact(in1 := "Bazine".benzina_90, in2 := 0.0)
      wire#w1
      Coil( "Alarme".alarme_vect[14] )
   END_RUNG
   RUNG wire#powerrail
      { S7_Templates := "SrcType := Real" } EQ_Contact(in1 := "Bazine".benzina_95, in2 := 0.0)
   END_RUNG wire#w1
   RUNG wire#powerrail
      { S7_Templates := "SrcType := Real" } EQ_Contact(in1 := "Bazine".motorina, in2 := 0.0)
   END_RUNG wire#w1
   RUNG wire#powerrail
      { S7_Templates := "SrcType := Real" } EQ_Contact(in1 := "Bazine".motorina_premium, in2 := 0.0)
   END_RUNG wire#w1
   // the same network as SCL:
   "Alarme".alarme_vect[14] := ("Bazine".benzina_90 = 0.0) OR ("Bazine".benzina_95 = 0.0) OR ("Bazine".motorina = 0.0) OR ("Bazine".motorina_premium = 0.0);
END_REGION

REGION Network 17: esd
   RUNG wire#powerrail
      Contact( "Avarii".esd_btn )
      Coil( "Alarme".alarme_vect[0] )
      Coil( "Avarii".esd )
   END_RUNG
   // the same network as SCL:
   "Alarme".alarme_vect[0] := "Avarii".esd_btn;
   "Avarii".esd := "Avarii".esd_btn;
END_REGION

REGION Network 18: reset esd
   IF "Avarii".reset_esd THEN "Avarii".esd_btn := FALSE; END_IF;
   "reset_esd".TON(IN := "Avarii".reset_esd, PT := T#3s);
   IF "reset_esd".Q THEN "Avarii".reset_esd := FALSE; END_IF;
END_REGION

REGION Network 19: avarii pe pompe
   RUNG wire#powerrail
      Contact( "Avarii".avarie_p1 )
      Coil( "Alarme".alarme_vect[1] )
   END_RUNG
   RUNG wire#powerrail
      Contact( "Avarii".avarie_p2 )
      Coil( "Alarme".alarme_vect[2] )
   END_RUNG
   RUNG wire#powerrail
      Contact( "Avarii".avarie_p3 )
      Coil( "Alarme".alarme_vect[3] )
   END_RUNG
   RUNG wire#powerrail
      Contact( "Avarii".avarie_p4 )
      Coil( "Alarme".alarme_vect[4] )
   END_RUNG
   // the same network as SCL:
   "Alarme".alarme_vect[1] := "Avarii".avarie_p1;
   "Alarme".alarme_vect[2] := "Avarii".avarie_p2;
   "Alarme".alarme_vect[3] := "Avarii".avarie_p3;
   "Alarme".alarme_vect[4] := "Avarii".avarie_p4;
END_REGION

REGION Network 20: reset avarii pe pompe
   IF "Avarii".reset_avarii AND "Avarii".avarie_p1 THEN "Avarii".avarie_p1 := FALSE; END_IF;
   IF "Avarii".reset_avarii AND "Avarii".avarie_p2 THEN "Avarii".avarie_p2 := FALSE; END_IF;
   IF "Avarii".reset_avarii AND "Avarii".avarie_p3 THEN "Avarii".avarie_p3 := FALSE; END_IF;
   IF "Avarii".reset_avarii AND "Avarii".avarie_p4 THEN "Avarii".avarie_p4 := FALSE; END_IF;
   "reset_avarii".TON(IN := "Avarii".reset_avarii, PT := T#3s);
   IF "reset_avarii".Q THEN "Avarii".reset_avarii := FALSE; END_IF;
END_REGION
END_ORGANIZATION_BLOCK

ORGANIZATION_BLOCK "Cyclic interrupt"   // OB30, LAD, CyclicInterrupt
{ S7_Optimized_Access := 'TRUE' }
VERSION : 0.1
   VAR_INPUT
      Initial_Call : Bool;   // Initial call of this OB
      Event_Count : Int;   // Events discarded
   END_VAR
BEGIN

REGION Network 1
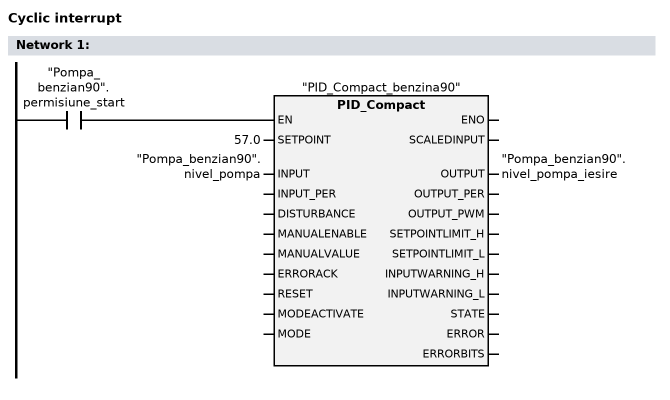
   IF "Pompa_benzian90".permisiune_start THEN
       "PID_Compact_benzina90"(Setpoint := 57.0,   // PID_Compact
                               Input := "Pompa_benzian90".nivel_pompa,
                               Output => "Pompa_benzian90".nivel_pompa_iesire);
   END_IF;
END_REGION
END_ORGANIZATION_BLOCK